INTERFACE ITF_Component1_HMI_Connector_Command EXTENDS ITF_BaseComponent_HMI_Connector_Command

END_INTERFACE

(* stored: Version 1.1.0.1
   Itf ITF_Component1_HMI_Connector_Command: Id {0cde79e7-27c3-02bf-3fff-9859f9c163a4} *)
